# B&R Automation Studio project appMain
Automation Studio 4.9.2.46; Test application

## Configuration FirstConfig

### Task classes (Cpu.sw)
```
Cyclic#1:
  MainPrg <- MainPrg.prg
  Program <- Application1.Program.prg
```

## Configuration SecondConfig

### Task classes (Cpu.sw)
```
Cyclic#4:
  Program <- Application1.Program.prg
  Program1 <- Application2.Program.prg
  MainPrg <- MainPrg.prg
```

## Logical view

### Global.var - Global variables
```iecst
VAR RETAIN
	machineName : STRING[255] := 'Machine2'; (*Name of the machine*)
END_VAR
```

### Program Logical/MainPrg (IEC)

#### Main.st
```iecst
PROGRAM _INIT

END_PROGRAM

PROGRAM _CYCLIC

END_PROGRAM

PROGRAM _EXIT

END_PROGRAM
```

Listed in the project but not available here: Logical/Global.typ, Logical/Libraries, Logical/Application1, Logical/Application2
